// TwinCAT 3 PLC project SubSysPLC
// ProgramVersion: 3.1.4022.7
// libraries:
//   Tc2_MC2, * (Beckhoff Automation GmbH)
//   Tc2_Standard, * (Beckhoff Automation GmbH)
//   Tc2_System, * (Beckhoff Automation GmbH)
//   Tc2_Utilities, * (Beckhoff Automation GmbH)
//   Tc3_Module, * (Beckhoff Automation GmbH)
//   PMPS,0.0.0,SLAC - LCLS
// project tree:
//   DUTs/ ST_BinarySolidAttenuator.TcDUT, ST_SolidAttenuatorBlade.TcDUT
//   GVLs/ GVL.TcGVL
//   / PlcTask.TcTTO
//   POUs/DatabaseComponents/ FB_ExampleDeviceSM_DB.TcPOU, FB_MySQL_Client.TcPOU, F_DB_To_hTable.TcPOU
//   POUs/DeviceImplementationEx1/ FB_ExampleDevice.TcPOU, FB_ExampleDeviceSM.TcPOU
//   POUs/DeviceImplementationEx2/ FB_DevMover.TcPOU, FB_ExampleDeviceSM_All.TcPOU
//   POUs/ Fast_Faults_Evaluate.TcPOU, MAIN.TcPOU, PMPS.TcPOU
// real-time tasks:
//   TASK PlcTask: cycle T#10ms, priority 20, ADS port 350
// motion (NC):
//   TASK NC-Task 1 SAF: cycle T#2ms, priority 4, ADS port 501
//   TASK NC-Task 1 SVB: cycle T#10ms, priority 8, ADS port 511
//   AXIS DevRunner_1 (id 3)
//     OtherSettings: AllowMotionCmdToSlave=true
//     encoder EncType=1
//     drive DrvType=5
//       Analog: ScaleFactorActTorque=0.1
//     controller CtrType=1
//       CtrPara: PriorControlFactor=1
//         Observer: BandWidth=20
//   AXIS DevRunner_2 (id 4)
//     OtherSettings: AllowMotionCmdToSlave=true
//     encoder EncType=1
//     drive DrvType=5
//       Analog: ScaleFactorActTorque=0.1
//     controller CtrType=1
//       CtrPara: PriorControlFactor=1
//         Observer: BandWidth=20
//   AXIS DevRunner_3 (id 5)
//     OtherSettings: AllowMotionCmdToSlave=true
//     encoder EncType=1
//     drive DrvType=5
//       Analog: ScaleFactorActTorque=0.1
//     controller CtrType=1
//       CtrPara: PriorControlFactor=1
//         Observer: BandWidth=20
//   AXIS DevRunner_4 (id 6)
//     OtherSettings: AllowMotionCmdToSlave=true
//     encoder EncType=1
//     drive DrvType=5
//       Analog: ScaleFactorActTorque=0.1
//     controller CtrType=1
//       CtrPara: PriorControlFactor=1
//         Observer: BandWidth=20
//   AXIS DevRunner_5 (id 7)
//     OtherSettings: AllowMotionCmdToSlave=true
//     encoder EncType=1
//     drive DrvType=5
//       Analog: ScaleFactorActTorque=0.1
//     controller CtrType=1
//       CtrPara: PriorControlFactor=1
//         Observer: BandWidth=20
//   AXIS DevRunner_6 (id 8)
//     OtherSettings: AllowMotionCmdToSlave=true
//     encoder EncType=1
//     drive DrvType=5
//       Analog: ScaleFactorActTorque=0.1
//     controller CtrType=1
//       CtrPara: PriorControlFactor=1
//         Observer: BandWidth=20
//   AXIS DevRunner_7 (id 9)
//     OtherSettings: AllowMotionCmdToSlave=true
//     encoder EncType=1
//     drive DrvType=5
//       Analog: ScaleFactorActTorque=0.1
//     controller CtrType=1
//       CtrPara: PriorControlFactor=1
//         Observer: BandWidth=20
//   AXIS DevRunner_8 (id 10)
//     OtherSettings: AllowMotionCmdToSlave=true
//     encoder EncType=1
//     drive DrvType=5
//       Analog: ScaleFactorActTorque=0.1
//     controller CtrType=1
//       CtrPara: PriorControlFactor=1
//         Observer: BandWidth=20
//   AXIS Dev1 (id 1)
//     OtherSettings: AllowMotionCmdToSlave=true
//     encoder EncType=1
//     drive DrvType=5
//       Analog: ScaleFactorActTorque=0.1
//     controller CtrType=1
//       CtrPara: PriorControlFactor=1
//         Observer: BandWidth=20
//   AXIS Dev2 (id 2)
//     OtherSettings: AllowMotionCmdToSlave=true
//     encoder EncType=1
//     drive DrvType=5
//       Analog: ScaleFactorActTorque=0.1
//     controller CtrType=1
//       CtrPara: PriorControlFactor=1
//         Observer: BandWidth=20
// I/O:
//   DEVICE Device 1 (EtherCAT), AmsNetId 0.0.0.0.2.1
//     Term 3 (EK1200) [EK1200-5000 EtherCAT Power supply (2A E-Bus)]
//       PMPS_FFO [EL2202 2Ch. Dig. Output 24V, 0.5A]
//       PMPS_PRE [EL6692 EtherCAT Bridge terminal (Primary)]
// variable links:
//   SubSysPLC Instance <-> Device 1 (EtherCAT)/Term 3 (EK1200)/PMPS_FFO
//     PlcTask Outputs/GVL.g_FastFaultOutput1.q_xFastFaultOut <-> Channel 1/Output
//   SubSysPLC Instance <-> Device 1 (EtherCAT)/Term 3 (EK1200)/PMPS_PRE
//     PlcTask Inputs/PMPS.fbArbiterIO.i_stCurrentBP <-> IO Inputs/CurrentBP
//     PlcTask Inputs/PMPS.fbArbiterIO.xTxPDO_state <-> SYNC Inputs/TxPDO state
//     PlcTask Inputs/PMPS.fbArbiterIO.xTxPDO_toggle <-> SYNC Inputs/TxPDO toggle
//     PlcTask Outputs/PMPS.fbArbiterIO.q_stRequestedBP <-> IO Outputs/RequestedBP
//   SubSysPLC Instance <-> NC-Task 1 SAF/Axes/Dev1
//     PlcTask Inputs/MAIN.fbDev1.stDevice.stAxis.NcToPlc <-> Outputs/ToPlc
//     PlcTask Outputs/MAIN.fbDev1.stDevice.stAxis.PlcToNc <-> Inputs/FromPlc
//   SubSysPLC Instance <-> NC-Task 1 SAF/Axes/Dev2
//     PlcTask Inputs/MAIN.fbDev2.stDevice.stAxis.NcToPlc <-> Outputs/ToPlc
//     PlcTask Outputs/MAIN.fbDev2.stDevice.stAxis.PlcToNc <-> Inputs/FromPlc
//   SubSysPLC Instance <-> NC-Task 1 SAF/Axes/DevRunner_1
//     PlcTask Inputs/MAIN.DevArray[1].stDevice.stAxis.NcToPlc <-> Outputs/ToPlc
//     PlcTask Outputs/MAIN.DevArray[1].stDevice.stAxis.PlcToNc <-> Inputs/FromPlc
//   SubSysPLC Instance <-> NC-Task 1 SAF/Axes/DevRunner_2
//     PlcTask Inputs/MAIN.DevArray[2].stDevice.stAxis.NcToPlc <-> Outputs/ToPlc
//     PlcTask Outputs/MAIN.DevArray[2].stDevice.stAxis.PlcToNc <-> Inputs/FromPlc
//   SubSysPLC Instance <-> NC-Task 1 SAF/Axes/DevRunner_3
//     PlcTask Inputs/MAIN.DevArray[3].stDevice.stAxis.NcToPlc <-> Outputs/ToPlc
//     PlcTask Outputs/MAIN.DevArray[3].stDevice.stAxis.PlcToNc <-> Inputs/FromPlc
//   SubSysPLC Instance <-> NC-Task 1 SAF/Axes/DevRunner_4
//     PlcTask Inputs/MAIN.DevArray[4].stDevice.stAxis.NcToPlc <-> Outputs/ToPlc
//     PlcTask Outputs/MAIN.DevArray[4].stDevice.stAxis.PlcToNc <-> Inputs/FromPlc
//   SubSysPLC Instance <-> NC-Task 1 SAF/Axes/DevRunner_5
//     PlcTask Inputs/MAIN.DevArray[5].stDevice.stAxis.NcToPlc <-> Outputs/ToPlc
//     PlcTask Outputs/MAIN.DevArray[5].stDevice.stAxis.PlcToNc <-> Inputs/FromPlc
//   SubSysPLC Instance <-> NC-Task 1 SAF/Axes/DevRunner_6
//     PlcTask Inputs/MAIN.DevArray[6].stDevice.stAxis.NcToPlc <-> Outputs/ToPlc
//     PlcTask Outputs/MAIN.DevArray[6].stDevice.stAxis.PlcToNc <-> Inputs/FromPlc
//   SubSysPLC Instance <-> NC-Task 1 SAF/Axes/DevRunner_7
//     PlcTask Inputs/MAIN.DevArray[7].stDevice.stAxis.NcToPlc <-> Outputs/ToPlc
//     PlcTask Outputs/MAIN.DevArray[7].stDevice.stAxis.PlcToNc <-> Inputs/FromPlc
//   SubSysPLC Instance <-> NC-Task 1 SAF/Axes/DevRunner_8
//     PlcTask Inputs/MAIN.DevArray[8].stDevice.stAxis.NcToPlc <-> Outputs/ToPlc
//     PlcTask Outputs/MAIN.DevArray[8].stDevice.stAxis.PlcToNc <-> Inputs/FromPlc

CONFIGURATION SubSysPLC
    RESOURCE PLC ON TwinCAT3
        TASK PlcTask(INTERVAL := T#10ms, PRIORITY := 20);
        PROGRAM MAIN WITH PlcTask : MAIN;
    END_RESOURCE
END_CONFIGURATION

// ---- DUTs/ST_BinarySolidAttenuator.TcDUT
TYPE ST_BinarySolidAttenuator :
STRUCT
	axBlades	: ARRAY [0..9] OF ST_SolidAttenuatorBlade;
END_STRUCT
END_TYPE

// ---- DUTs/ST_SolidAttenuatorBlade.TcDUT
TYPE ST_SolidAttenuatorBlade :
STRUCT
	xRequestedIn	:	BOOL;
	xCurrentIn	:	BOOL;
	rThickness	:	REAL;
END_STRUCT
END_TYPE

// ---- GVLs/GVL.TcGVL

VAR_GLOBAL
	g_fbArbiter1	:	FB_Arbiter;
	g_fbArbiter2	:	FB_Arbiter;
	{attribute 'TcLinkTo' := '.q_xFastFaultOut:=TIIB[PMPS_FFO]^Channel 1^Output'}
	g_FastFaultOutput1	:	FB_HardwareFFOutput;
	g_rTestingVelocity	:	LREAL := PMPS_GVL.VISIBLE_TEST_VELOCITY;
END_VAR

// ---- POUs/MAIN.TcPOU
PROGRAM MAIN
VAR
	fbDev1	:	FB_ExampleDeviceSM_All;
	fbDev1Mover	:	FB_DevMover;
	fbDev2	:	FB_ExampleDeviceSM_All;
	fbDev2Mover	:	FB_DevMover;
	
	rtInit	:	R_TRIG;
	Initialize	:	BOOL := TRUE;
	
	DevArray : ARRAY[1..8] OF FB_ExampleDeviceSM_All;
	DevMoverArray : ARRAY [1..8] OF FB_DevMover;
	
	//fbDev3	:	FB_ExampleDeviceSM_DB;

	DevRunnerInt: INT;
	
	AttemptReset	:	TON;
    
    ffArray : ARRAY[1..FF_ARRAY] OF FB_FastFault;
    FFRunnerInt : INT := 1;
END_VAR
VAR CONSTANT
    FF_ARRAY : INT := 200;
END_VAR

//Sub-system Device PLC

IF Initialize THEN
	fbDev1(cBase := 10,
		fbFastFaultOutput := g_FastFaultOutput1,
		fbArbiter := g_fbArbiter1);
	fbDev2(cBase := 1000,
		fbFastFaultOutput := g_FastFaultOutput1,
		fbArbiter := g_fbArbiter1);
	g_fbArbiter1.A_Init();

//	fbDev3(cBase := 0,iDBID:=1,sDBNetId:='172.21.42.53.1.1',sDeviceID:='1',
//		fbArbiter := g_fbArbiter,
//		fbFastFaultOutput := g_FastFaultOutput1);

	FOR DevRunnerInt := 1 TO 8 DO
		DevArray[DevRunnerInt](cBase := DevRunnerInt*1000,
			fbFastFaultOutput := g_FastFaultOutput1,
			fbArbiter := g_fbArbiter1);
	END_FOR

	Initialize := FALSE;
END_IF

//Example devices
fbDev1(fbFastFaultOutput := g_FastFaultOutput1,
		fbArbiter := g_fbArbiter1);
fbDev2(fbFastFaultOutput := g_FastFaultOutput1,
		fbArbiter := g_fbArbiter1);
		
fbDev1Mover(Device:=fbDev1.stDevice);
fbDev2Mover(Device:=fbDev2.stDevice);

FOR DevRunnerInt := 1 TO 8 DO
	DevArray[DevRunnerInt](cBase := DevRunnerInt*1000,
		fbFastFaultOutput := g_FastFaultOutput1,
		fbArbiter := g_fbArbiter1);
		
	DevMoverArray[DevRunnerInt](Device := DevArray[DevRunnerInt].stDevice);	
END_FOR
(*
FOR FFRunnerInt := 1 to FF_ARRAY DO
    ffArray[FFRunnerInt](io_fbFFHWO := g_FastFaultOutput1);
END_FOR
*)		
PMPS();

Fast_Faults_Evaluate();

ACTION Initialize:

END_ACTION

END_PROGRAM

// ---- POUs/DeviceImplementationEx2/FB_ExampleDeviceSM_All.TcPOU
(* This version of the block is self contained. Minimizes wiring.*)
FUNCTION_BLOCK FB_ExampleDeviceSM_All
VAR_INPUT
	cBase: UDINT;
END_VAR
VAR_OUTPUT
END_VAR
VAR_IN_OUT
	fbFastFaultOutput	:	FB_HardwareFFOutput;
	fbArbiter	:	FB_Arbiter;
END_VAR
VAR
	stDevice	:	ST_Device;
	fbGovernor	:	FB_LinearGovernor;
	mcPower	:	MC_Power;
	mcStop: MC_Stop;
	mcAbsolute	:	MC_MoveAbsolute;
	fbBPTM	:	BeamParameterTransitionManager;
	xStartMove: BOOL;
	
	stCheckState: ST_DeviceState;
	stTargetState	:	ST_DeviceState; //Target device state

END_VAR
VAR PERSISTENT
	nLastActiveState	:	UDINT;
END_VAR

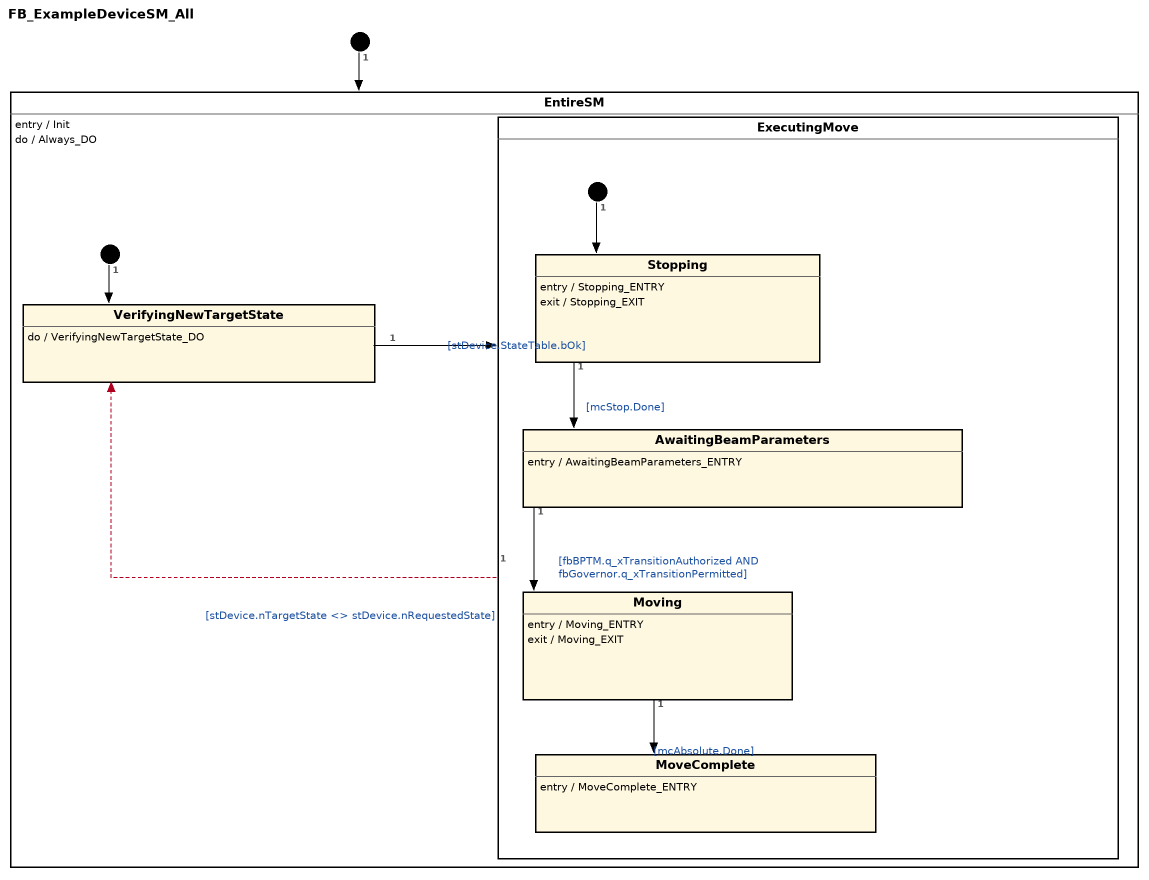
STATECHART FB_ExampleDeviceSM_All_1  // abortable
    START StartState3
    COMPOSITE STATE EntireSM
        entry / Init
        do / Always_DO
        START StartState1
        COMPOSITE STATE ExecutingMove
            START StartState2
            STATE Stopping
                entry / Stopping_ENTRY
                exit / Stopping_EXIT
            STATE AwaitingBeamParameters
                entry / AwaitingBeamParameters_ENTRY
            STATE Moving
                entry / Moving_ENTRY
                exit / Moving_EXIT
            STATE MoveComplete
                entry / MoveComplete_ENTRY
            StartState2 -> Stopping  // priority 1, on completion
            Stopping -> AwaitingBeamParameters [mcStop.Done] // priority 1, rising edge
            AwaitingBeamParameters -> Moving [fbBPTM.q_xTransitionAuthorized AND fbGovernor.q_xTransitionPermitted] // priority 1, rising edge
            Moving -> MoveComplete [mcAbsolute.Done] // priority 1, rising edge
        END_STATE
        STATE VerifyingNewTargetState
            do / VerifyingNewTargetState_DO
        StartState1 -> VerifyingNewTargetState  // priority 1, on completion
        ExecutingMove -> VerifyingNewTargetState [stDevice.nTargetState <> stDevice.nRequestedState] // priority 1, exception, rising edge
        VerifyingNewTargetState -> ExecutingMove [stDevice.StateTable.bOk] // priority 1
    END_STATE
    StartState3 -> EntireSM  // priority 1, on completion
END_STATECHART

ACTION Always_DO:
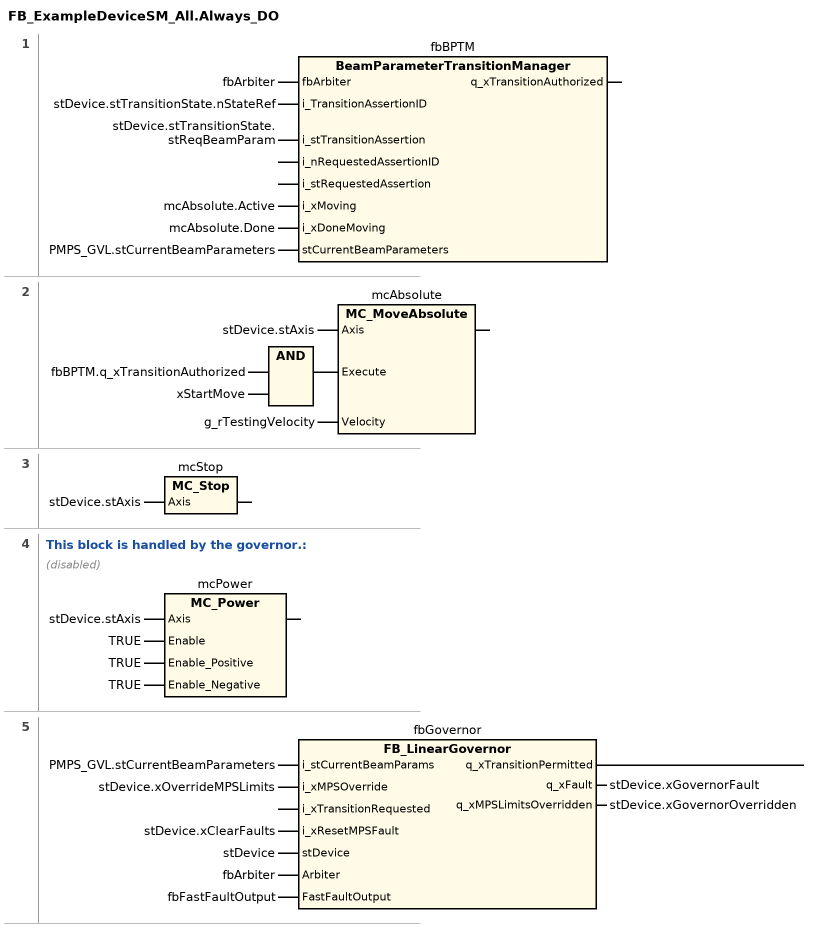
// NETWORK 1
fbBPTM(
    fbArbiter := fbArbiter,
    i_TransitionAssertionID := stDevice.stTransitionState.nStateRef,
    i_stTransitionAssertion := stDevice.stTransitionState.stReqBeamParam,
    i_xMoving := mcAbsolute.Active,
    i_xDoneMoving := mcAbsolute.Done,
    stCurrentBeamParameters := PMPS_GVL.stCurrentBeamParameters); // BeamParameterTransitionManager

// NETWORK 2
mcAbsolute(
    Axis := stDevice.stAxis,
    Execute := fbBPTM.q_xTransitionAuthorized AND xStartMove,
    Velocity := g_rTestingVelocity); // MC_MoveAbsolute

// NETWORK 3
mcStop(Axis := stDevice.stAxis); // MC_Stop

// NETWORK 4 (disabled)
// label: This block is handled by the governor.
// mcPower(Axis := stDevice.stAxis, Enable := TRUE, Enable_Positive := TRUE, Enable_Negative := TRUE); // MC_Power

// NETWORK 5
fbGovernor(
    i_stCurrentBeamParams := PMPS_GVL.stCurrentBeamParameters,
    i_xMPSOverride := stDevice.xOverrideMPSLimits,
    i_xResetMPSFault := stDevice.xClearFaults,
    stDevice := stDevice,
    Arbiter := fbArbiter,
    FastFaultOutput := fbFastFaultOutput,
    q_xFault => stDevice.xGovernorFault,
    q_xMPSLimitsOverridden => stDevice.xGovernorOverridden); // FB_LinearGovernor
END_ACTION

ACTION AwaitingBeamParameters_ENTRY:
fbBPTM.i_stRequestedAssertion := stTargetState.stReqBeamParam;
fbBPTM.i_nRequestedAssertionID := stTargetState.nStateRef;

//Tell the governor that we're trying to move.
fbGovernor.i_xTransitionRequested := TRUE;
END_ACTION

ACTION Init:

//Safe State
stDevice.nSafeState := cBase;
stDevice.nTransitionState := cBase+100;

//Initialize the State Table
stDevice.StateTable.A_Reset();

//Device State Table Instantiation
//To be done by the device state table database system
F_SetStateParams(
	nStateRef := stDevice.nSafeState,
	rPosition := 0,
	rTolerance := 10,
	stBeamParams := PMPS_GVL.cstFullBeam,
	Table := stDevice.StateTable
);
F_SetStateParams(
	nStateRef := cBase + 1,
	rPosition := 100,
	rTolerance := 10,
	stBeamParams := F_SetBeamParams(
		fAtt := 20,
		fPP_mJ := 1,
		neVRange	:= 2#1111_1011_1111_0000,
		nRate := 10
		),
	Table := stDevice.StateTable
);
F_SetStateParams(
	nStateRef := cBase + 2,
	rPosition := 200,
	rTolerance := 10,
	stBeamParams := F_SetBeamParams(
		fAtt := 30,
		fPP_mJ := 1,
		neVRange	:= 2#1111_1011_1111_0000,
		nRate := 10
		),
	Table := stDevice.StateTable
);
F_SetStateParams(
	nStateRef := cBase + 3,
	rPosition := 300,
	rTolerance := 10,
	stBeamParams := F_SetBeamParams(
		fAtt := 20,
		fPP_mJ := 1,
		neVRange	:= 2#1111_1011_1111_0000,
		nRate := 10
		),
	Table := stDevice.StateTable
);

F_SetStateParams(
	nStateRef := stDevice.nTransitionState,
	rPosition := 0,
	rTolerance := 0,
	stBeamParams := F_SetBeamParams(
		fAtt := 0,
		fPP_mJ := 0,
		neVRange	:= 2#1111_1011_1111_0000,
		nRate := 0
		),
	Table := stDevice.StateTable
);

//Set device transition state
stDevice.StateTable.A_Lookup(
	key := stDevice.nTransitionState,
	getValue => stDevice.stTransitionState
);

//Need an initialization routine for setting the active state
//Check if the device is at safe state
//If the device is within the state boundaries, it's considered to be in that state
stDevice.StateTable.A_Lookup(key:= stDevice.nSafeState);
IF stDevice.StateTable.bOk THEN
	stCheckState := stDevice.StateTable.getValue;
ELSE
	stCheckState := stDevice.stTransitionState; //This needs to be safer <TODO>
END_IF

IF stDevice.stAxis.NcToPlc.ActPos <= stCheckstate.rPosition + stCheckState.rTolerance AND
	stDevice.stAxis.NcToPlc.ActPos >= stCheckState.rPosition - stCheckState.rTolerance THEN
	stDevice.nActiveState := nLastActiveState;
ELSE
	stDevice.nActiveState := stDevice.nTransitionState;
END_IF

//Simulation Hardware Limit Switches
stDevice.i_xHiLim := TRUE;
stDevice.i_xLoLim := TRUE;
END_ACTION

ACTION MoveComplete_ENTRY:
//Clear transition request
fbGovernor.i_xTransitionRequested := FALSE;
//Latch active state
stDevice.nActiveState := stDevice.nTargetState;
nLastActiveState := stDevice.nActiveState;
END_ACTION

ACTION Moving_ENTRY:
xStartMove := TRUE;
mcAbsolute.Position := stTargetState.rPosition;
END_ACTION

ACTION Moving_EXIT:
xStartMove := FALSE;
END_ACTION

ACTION NewMove_ENTRY:

END_ACTION

ACTION Stopping_ENTRY:
mcStop.Execute := TRUE;
END_ACTION

ACTION Stopping_EXIT:
mcStop.Execute := FALSE;
END_ACTION

ACTION VerifyingNewTargetState_DO:
stDevice.StateTable.A_Lookup(
	key := stDevice.nRequestedState
);

IF stDevice.StateTable.bOk THEN
	stTargetState := stDevice.StateTable.getValue;
	stDevice.nTargetState := stDevice.nRequestedState;
ELSE
	; //log ignored state/ generate an error? <TODO>
END_IF
END_ACTION

END_FUNCTION_BLOCK

// ---- POUs/DeviceImplementationEx2/FB_DevMover.TcPOU
FUNCTION_BLOCK FB_DevMover
VAR_IN_OUT
	Device: ST_Device;
END_VAR

VAR
	DevMoverState: INT := 0;
	getPosPtr    : POINTER TO PMPS.T_HashTableEntry := 0;(* Returned hash table entry position pointer *)
	Pause : TON := (PT := T#5s);
	StartAgain: R_TRIG;
	Restart: BOOL;
END_VAR


StartAgain(CLK:=Restart);
Restart R= StartAgain.Q;
IF StartAgain.Q THEN
	DevMoverState := 0;
END_IF

CASE DevMoverState OF
	0:
		DevMoverState := 100;
	100: //Go to first entry in the state table
		Device.StateTable.A_GetFirst();
		//Device.nRequestedState := Device.StateTable.getValue.nStateRef;
		getPosPtr := Device.StateTable.getPosPtr;
		// Wait for move to complete
		DevMoverState := 300;
		
	200: // Wait for move
		
		// Once move is done, go to next entry in state table
		Pause(IN := Device.nActiveState = Device.nTargetState);
		IF Pause.Q THEN
			DevMoverState := 300;
		END_IF
(*		
	250: // Move to upper limit
	
	251: // Move to lower limit
*)	
	300: // Go to next entry
		Device.StateTable.A_GetNext(putPosPtr:=getPosPtr);
		
		// Go back to wait for move unless there are no more entries
		IF Device.StateTable.bOk AND (Device.StateTable.getValue.nStateRef <> Device.nRequestedState) THEN
			Device.nRequestedState := Device.StateTable.getValue.nStateRef;
			getPosPtr := Device.StateTable.getPosPtr;
			DevMoverState := 200;
		ELSE
			DevMoverState := 100;
		END_IF
		
	
END_CASE

END_FUNCTION_BLOCK

// ---- POUs/PMPS.TcPOU
PROGRAM PMPS
VAR
    
    fbArbiterIO : FB_SubSysToArbiter_IO;
END_VAR

fbArbiterIO(Arbiter := GVL.g_fbArbiter1, fbFFHWO := GVL.g_FastFaultOutput1);

END_PROGRAM

// ---- POUs/Fast_Faults_Evaluate.TcPOU
PROGRAM Fast_Faults_Evaluate
VAR
END_VAR

g_FastFaultOutput1.EvaluateOutput();

END_PROGRAM

// ---- POUs/DatabaseComponents/FB_ExampleDeviceSM_DB.TcPOU
(* This version of the block is self contained. Minimizes wiring.*)
FUNCTION_BLOCK FB_ExampleDeviceSM_DB
VAR_INPUT
	cBase: UDINT;
	iDBID:UDINT;
	sDBNetId: STRING;
	sDeviceID: STRING;
END_VAR
VAR_OUTPUT
END_VAR
VAR_IN_OUT
	fbArbiter : FB_Arbiter;
	fbFastFaultOutput	:	FB_HardwareFFOutput;
END_VAR
VAR
	stDevice	:	ST_Device;
	fbGovernor	:	FB_LinearGovernor;
	mcPower	:	MC_Power;
	mcStop: MC_Stop;
	mcAbsolute	:	MC_MoveAbsolute;
	fbBPTM	:	BeamParameterTransitionManager;
	xStartMove: BOOL;
	
	stCheckState: ST_DeviceState;
	stTargetState	:	ST_DeviceState; //Target device state
	fbDBClient:FB_MySQL_Client;
	bInitReady: BOOL :=FALSE;
	//aStateTable : ARRAY[1..PMPS_GVL.MAX_DEVICE_STATES] OF ST_DeviceStateTable;

END_VAR
VAR PERSISTENT
	nLastActiveState	:	UDINT;
END_VAR

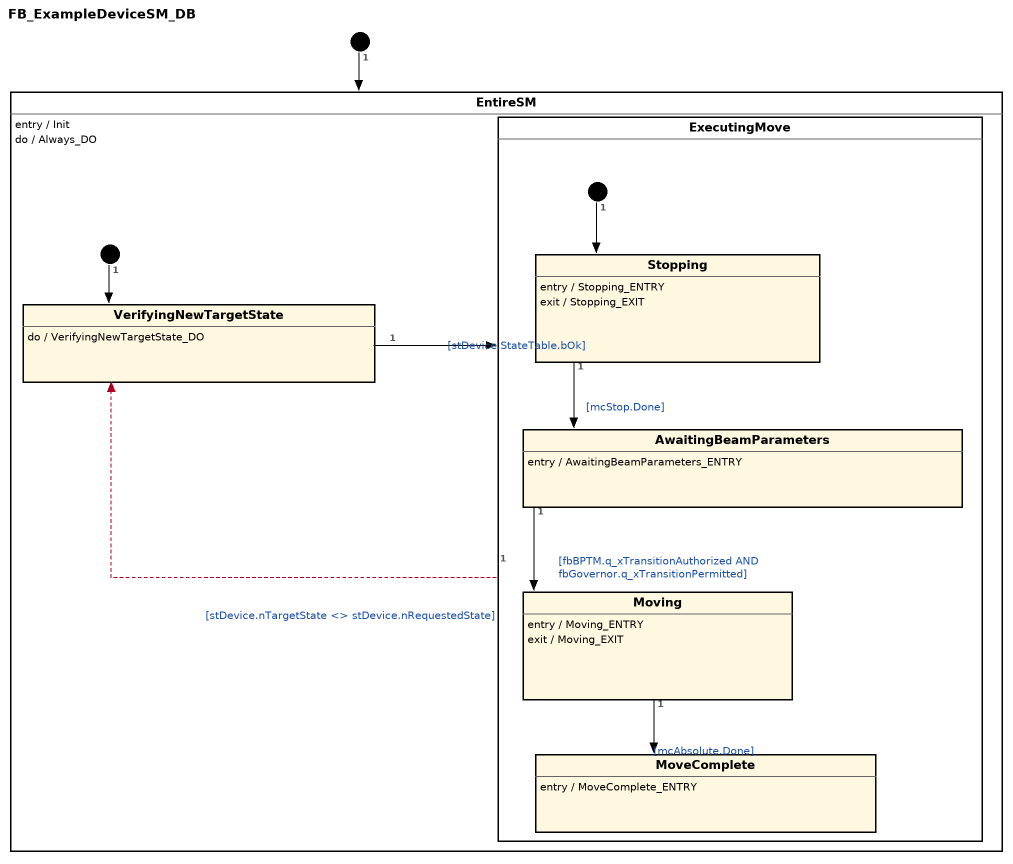
STATECHART FB_ExampleDeviceSM_DB  // abortable
    START StartState3
    COMPOSITE STATE EntireSM
        entry / Init
        do / Always_DO
        START StartState1
        COMPOSITE STATE ExecutingMove
            START StartState2
            STATE Stopping
                entry / Stopping_ENTRY
                exit / Stopping_EXIT
            STATE AwaitingBeamParameters
                entry / AwaitingBeamParameters_ENTRY
            STATE Moving
                entry / Moving_ENTRY
                exit / Moving_EXIT
            STATE MoveComplete
                entry / MoveComplete_ENTRY
            StartState2 -> Stopping  // priority 1, on completion
            Stopping -> AwaitingBeamParameters [mcStop.Done] // priority 1, rising edge
            AwaitingBeamParameters -> Moving [fbBPTM.q_xTransitionAuthorized AND fbGovernor.q_xTransitionPermitted] // priority 1, rising edge
            Moving -> MoveComplete [mcAbsolute.Done] // priority 1, rising edge
        END_STATE
        STATE VerifyingNewTargetState
            do / VerifyingNewTargetState_DO
        StartState1 -> VerifyingNewTargetState  // priority 1, on completion
        ExecutingMove -> VerifyingNewTargetState [stDevice.nTargetState <> stDevice.nRequestedState] // priority 1, exception, rising edge
        VerifyingNewTargetState -> ExecutingMove [stDevice.StateTable.bOk] // priority 1
    END_STATE
    StartState3 -> EntireSM  // priority 1, on completion
END_STATECHART

ACTION Always_DO:
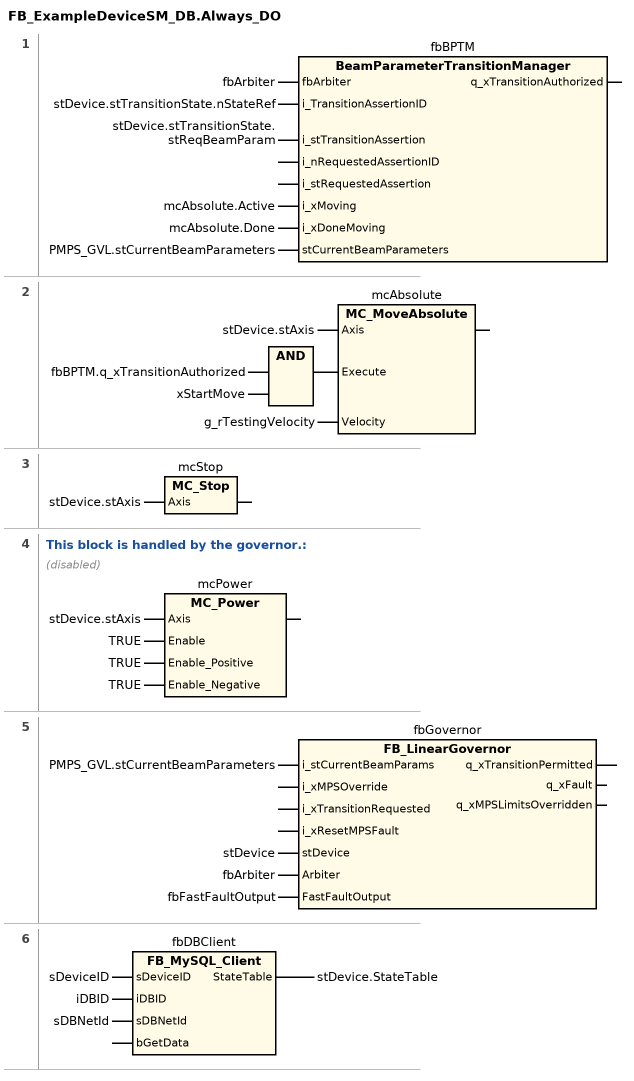
// NETWORK 1
fbBPTM(
    fbArbiter := fbArbiter,
    i_TransitionAssertionID := stDevice.stTransitionState.nStateRef,
    i_stTransitionAssertion := stDevice.stTransitionState.stReqBeamParam,
    i_xMoving := mcAbsolute.Active,
    i_xDoneMoving := mcAbsolute.Done,
    stCurrentBeamParameters := PMPS_GVL.stCurrentBeamParameters); // BeamParameterTransitionManager

// NETWORK 2
mcAbsolute(
    Axis := stDevice.stAxis,
    Execute := fbBPTM.q_xTransitionAuthorized AND xStartMove,
    Velocity := g_rTestingVelocity); // MC_MoveAbsolute

// NETWORK 3
mcStop(Axis := stDevice.stAxis); // MC_Stop

// NETWORK 4 (disabled)
// label: This block is handled by the governor.
// mcPower(Axis := stDevice.stAxis, Enable := TRUE, Enable_Positive := TRUE, Enable_Negative := TRUE); // MC_Power

// NETWORK 5
fbGovernor(
    i_stCurrentBeamParams := PMPS_GVL.stCurrentBeamParameters,
    stDevice := stDevice,
    Arbiter := fbArbiter,
    FastFaultOutput := fbFastFaultOutput); // FB_LinearGovernor

// NETWORK 6
fbDBClient(sDeviceID := sDeviceID, iDBID := iDBID, sDBNetId := sDBNetId); // FB_MySQL_Client
stDevice.StateTable := fbDBClient.StateTable;
END_ACTION

ACTION AwaitingBeamParameters_ENTRY:
fbBPTM.i_stRequestedAssertion := stTargetState.stReqBeamParam;
fbBPTM.i_nRequestedAssertionID := stTargetState.nStateRef;

//Tell the governor that we're trying to move.
fbGovernor.i_xTransitionRequested := TRUE;
END_ACTION

ACTION Init:
	
//Safe State
stDevice.nSafeState := cBase;
stDevice.nTransitionState := cBase+100;

//Initialize the State Table
stDevice.StateTable.A_Reset();
//Device State Table Instantiation
F_SetStateParams(
	nStateRef := stDevice.nSafeState,
	rPosition := 0,
	rTolerance := 10,
	stBeamParams := PMPS_GVL.cstFullBeam,
	Table := stDevice.StateTable
);
//Connect to DB and get state table data
fbDBClient.bGetData:= TRUE;//fbMySQL.nState:=400; 

stDevice.StateTable.A_Lookup(
		key := stDevice.nTransitionState,
		getValue => stDevice.stTransitionState
);
	
//Need an initialization routine for setting the active state
//Check if the device is at the last known state
//If the device is within the state boundaries, it's considered to be in that state
stDevice.StateTable.A_Lookup(key:= nLastActiveState);
IF stDevice.StateTable.bOk THEN
	stCheckState := stDevice.StateTable.getValue;
ELSE
	stCheckState := stDevice.stTransitionState; //This needs to be safer <TODO>
END_IF

IF stDevice.stAxis.NcToPlc.ActPos <= stCheckstate.rPosition + stCheckState.rTolerance AND
	stDevice.stAxis.NcToPlc.ActPos >= stCheckState.rPosition - stCheckState.rTolerance THEN
	stDevice.nActiveState := nLastActiveState;
ELSE
	stDevice.nActiveState := stDevice.nTransitionState;
END_IF

//Simulation Hardware Limit Switches
stDevice.i_xHiLim := TRUE;
stDevice.i_xLoLim := TRUE;
END_ACTION

ACTION Initialize:

END_ACTION

ACTION MoveComplete_ENTRY:
//Clear transition request
fbGovernor.i_xTransitionRequested := FALSE;
//Latch active state
stDevice.nActiveState := stDevice.nTargetState;
nLastActiveState := stDevice.nActiveState;
END_ACTION

ACTION Moving_ENTRY:
xStartMove := TRUE;
mcAbsolute.Position := stTargetState.rPosition;
END_ACTION

ACTION Moving_EXIT:
xStartMove := FALSE;
END_ACTION

ACTION NewMove_ENTRY:

END_ACTION

ACTION Stopping_ENTRY:
mcStop.Execute := TRUE;
END_ACTION

ACTION Stopping_EXIT:
mcStop.Execute := FALSE;
END_ACTION

ACTION VerifyingNewTargetState_DO:
stDevice.StateTable.A_Lookup(
	key := stDevice.nRequestedState
);

IF stDevice.StateTable.bOk THEN
	stTargetState := stDevice.StateTable.getValue;
	stDevice.nTargetState := stDevice.nRequestedState;
ELSE
	; //log ignored state/ generate an error? <TODO>
END_IF
END_ACTION

END_FUNCTION_BLOCK

// ---- POUs/DatabaseComponents/FB_MySQL_Client.TcPOU
FUNCTION_BLOCK FB_MySQL_Client
VAR_INPUT
	sDeviceID: STRING;
	iDBID:UDINT;
	sDBNetId: STRING ;
	bGetData:BOOL;
END_VAR
VAR_OUTPUT
	StateTable : FB_LinearDeviceStateTable;
END_VAR
VAR CONSTANT
	sSQLCommand :STRING:='SELECT * FROM device_states  WHERE device_id =';
END_VAR
VAR
	nState: INT:=0; // used as a start signal
	nRecordCount: UDINT:=PMPS_GVL.MAX_DEVICE_STATES;
	aDeviceStateTable : ARRAY[1..PMPS_GVL.MAX_DEVICE_STATES] OF ST_DeviceStateTable;
	fbMySQLDB:  FB_SQLDatabase(sNetId := '', tTimeout:=T#5S);
	fbSQLCmd:  FB_SQLCommand(sNetId := '', tTimeout:=T#5S);
	fbSQLResult: FB_SQLResult(sNetId := '', tTimeout:=T#5S);
	sSQLCmd :STRING;
	ipResultEvent : Tc3_Eventlogger.I_TcResultEvent;
	
	
END_VAR


IF (bGetData) THEN
	bGetData:= FALSE;
	nState := 100;
END_IF

CASE nState OF
	0:
100:// Initialize Database function blocks
	fbMySQLDB.sNetID := sDBNetId;
	fbSQLCmd.sNetID := sDBNetId;
	fbSQLResult.sNetID := sDBNetId; 
	IF fbMySQLDB.Connect(iDBID) THEN
		IF fbMySQLDB.bError THEN
			nState := 9000+nState; 
		ELSE
			nState := nState+1; 
		END_IF
	END_IF
 
101:	
	 IF(fbMySQLDB.bConnected ) THEN
		fbMySQLDB.CreateCmd(pSQLCommand := ADR(fbSQLCmd));
		IF fbMySQLDB.bError THEN
			nState := 9000+nState; 
		ELSE
			nState := 1+nState; 
		END_IF
	 END_IF
102:	 
  (*Execute SQL Comnmand*)
	//sSQLCmd :=sSQLCommand;
	sSQLCmd := CONCAT(sSQLCommand, sDeviceID) ;		
   IF fbSQLCmd.ExecuteDataReturn(pSQLCmd:=ADR(sSQLCmd),cbSQLCmd:=SIZEOF(sSQLCmd),pSQLDBResult:=ADR(fbSQLResult)) THEN
   	IF( fbSQLCmd.bError) THEN
	    nState := 9000+nState; 
    ELSE
        nState := 1+nState; 
		MEMSET(ADR(aDeviceStateTable),0,SIZEOF(aDeviceStateTable));

    END_IF
  END_IF
 
103: 
	(*Read data FROM the database*)
  IF (fbSQLResult.Read(nStartIndex:=0, nRecordCount:=nRecordCount,pData:=ADR(aDeviceStateTable),cbData:=SIZEOF(aDeviceStateTable),bWithVerifying:=TRUE,bDataRelease:=TRUE) )THEN
	 ipResultEvent := fbSQLResult.ipTcResultEvent;
	IF fbSQLResult.bError THEN
         nState := 9000+nState; 
    ELSE
        nState := 500;// 1+nState; 
    END_IF
END_IF	

500:
	//Device State Table Instantiation
	IF F_DB_To_hTable( aStatesParamsTable:= aDeviceStateTable, nRecordCount:=nRecordCount, Table := StateTable)THEN
         nState := 9000+nState; 
    ELSE
        nState :=800;// 1+nState; 
    END_IF



600: //Reload DATA
//Reset all hash table entries
// re instantiate device state table	
	;
9500:
800: //Release and Disconnect
	
	IF (fbSQLResult.Release() AND fbMySQLDB.Disconnect()) THEN
		nState:=-1;
		ELSE
			 nState := 9000+nState; 
	END_IF


		;
END_CASE

END_FUNCTION_BLOCK

// ---- POUs/DatabaseComponents/F_DB_To_hTable.TcPOU
FUNCTION F_DB_To_hTable : BOOL
VAR_INPUT
	aStatesParamsTable : ARRAY[1..PMPS_GVL.MAX_DEVICE_STATES] OF ST_DeviceStateTable;
	nRecordCount: UDINT;
END_VAR
VAR_IN_OUT
	Table	:	FB_LinearDeviceStateTable;
END_VAR
VAR
	stDeviceState	:	ST_DeviceState;
	iRow : UDINT:=1;
END_VAR

Table.A_Reset();
//Device State Table Instantiation
(*F_SetStateParams(
	nStateRef := 0,
	rPosition := 0,
	rTolerance := 0,
	stBeamParams := PMPS_GVL.cstFullBeam,
	Table := Table
);
*)
IF (nRecordCount>0) THEN
	FOR iRow:=1 TO nRecordCount BY 1 DO
	stDeviceState.nStateRef := DINT_TO_UDINT(aStatesParamsTable[iRow].iStateID);
	stDeviceState.rPosition := aStatesParamsTable[iRow].rTargetPosition;
	stDeviceState.rTolerance := aStatesParamsTable[iRow].rTolerance;  
	stDeviceState.stReqBeamParam.fAtt := aStatesParamsTable[iRow].rTransmission;
	stDeviceState.stReqBeamParam.fPP_mJ := (aStatesParamsTable[iRow].rPerPulseEnergy);
	stDeviceState.stReqBeamParam.nRate := DINT_TO_UDINT(aStatesParamsTable[iRow].iPulseRate);
	stDeviceState.stReqBeamParam.nBeamClass := DINT_TO_BYTE(aStatesParamsTable[iRow].iBeamClass);
//	stDeviceState.stReqBeamParam.fUpper_eV := (aStatesParamsTable[iRow].rUpper_eV);
//	stDeviceState.stReqBeamParam.fLower_eV := (aStatesParamsTable[iRow].rLower_eV);
	stDeviceState.stReqBeamParam.reV := aStatesParamsTable[iRow].rPhotonEnergy;
	//stDeviceState.stReqBeamParam.neVRange := (aStatesParamsTable[iRow].rLower_eV);
	Table.A_Add(
		key := stDeviceState.nStateRef,
		putValue := stDeviceState
	);
END_FOR;
END_IF

Table.A_Count();
F_DB_To_hTable := Table.bOk;

END_FUNCTION

// ---- POUs/DeviceImplementationEx1/FB_ExampleDevice.TcPOU
FUNCTION_BLOCK FB_ExampleDevice
VAR_INPUT
END_VAR
VAR_OUTPUT
END_VAR
VAR
	MC_MoveAbsolute_0: MC_MoveAbsolute;
	fbBCTM: BeamParameterTransitionManager;
	FB_ExampleDeviceSM_0: FB_ExampleDeviceSM;
	stDevice	:	ST_Device;
	MC_Power_0: MC_Power;
	MC_Stop_0	:	MC_Stop;
END_VAR

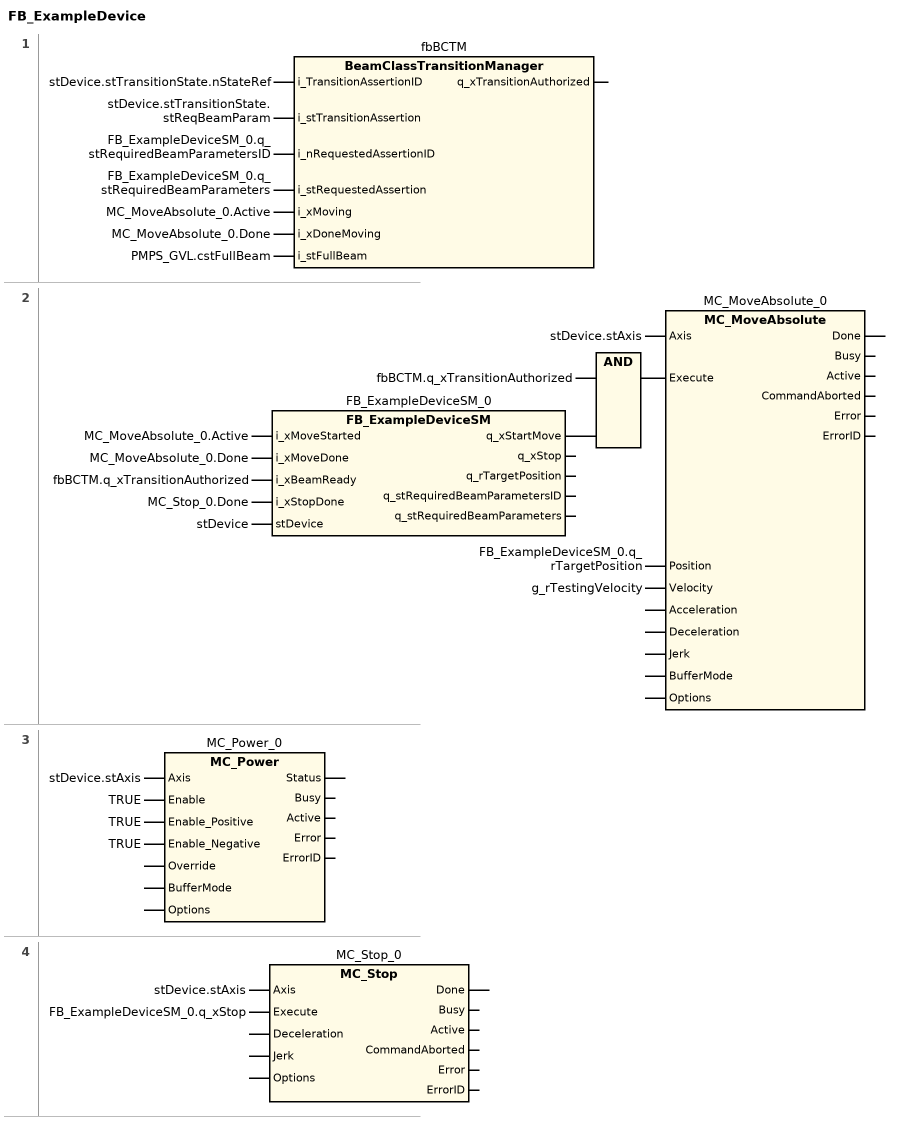
// NETWORK 1
fbBCTM(
    i_TransitionAssertionID := stDevice.stTransitionState.nStateRef,
    i_stTransitionAssertion := stDevice.stTransitionState.stReqBeamParam,
    i_nRequestedAssertionID := FB_ExampleDeviceSM_0.q_stRequiredBeamParametersID,
    i_stRequestedAssertion := FB_ExampleDeviceSM_0.q_stRequiredBeamParameters,
    i_xMoving := MC_MoveAbsolute_0.Active,
    i_xDoneMoving := MC_MoveAbsolute_0.Done,
    i_stFullBeam := PMPS_GVL.cstFullBeam); // BeamClassTransitionManager

// NETWORK 2
FB_ExampleDeviceSM_0(
    i_xMoveStarted := MC_MoveAbsolute_0.Active,
    i_xMoveDone := MC_MoveAbsolute_0.Done,
    i_xBeamReady := fbBCTM.q_xTransitionAuthorized,
    i_xStopDone := MC_Stop_0.Done,
    stDevice := stDevice); // FB_ExampleDeviceSM
MC_MoveAbsolute_0(
    Axis := stDevice.stAxis,
    Execute := fbBCTM.q_xTransitionAuthorized AND FB_ExampleDeviceSM_0.q_xStartMove,
    Position := FB_ExampleDeviceSM_0.q_rTargetPosition,
    Velocity := g_rTestingVelocity); // MC_MoveAbsolute

// NETWORK 3
MC_Power_0(Axis := stDevice.stAxis, Enable := TRUE, Enable_Positive := TRUE, Enable_Negative := TRUE); // MC_Power

// NETWORK 4
MC_Stop_0(Axis := stDevice.stAxis, Execute := FB_ExampleDeviceSM_0.q_xStop); // MC_Stop

ACTION Initialize:

stDevice.astStates[1].rPosition := 100;
stDevice.astStates[1].nStateRef := 16#1;
stDevice.astStates[1].stReqBeamParam := F_SetBeamParams(
	fAtt := 20,
	fPP_mJ := 1,
	fLower_eV := 0,
	fUpper_eV := 1500
);

stDevice.astStates[2].rPosition := 200;
stDevice.astStates[2].nStateRef := 16#2;
stDevice.astStates[2].stReqBeamParam := F_SetBeamParams(
	fAtt := 50,
	fPP_mJ := 1,
	fLower_eV := 0,
	fUpper_eV := 1500
);

stDevice.astStates[3].rPosition := 300;
stDevice.astStates[3].nStateRef := 16#3;
stDevice.astStates[3].stReqBeamParam := F_SetBeamParams(
	fAtt := 50,
	fPP_mJ := 0.5,
	fLower_eV := 0,
	fUpper_eV := 1500
);

stDevice.stTransitionState.nStateRef := 16#10;
stDevice.stTransitionState.stReqBeamParam := F_SetBeamParams(
	fAtt := 100,
	fPP_mJ := 1,
	fLower_eV := 0,
	fUpper_eV := 1500
);
END_ACTION

END_FUNCTION_BLOCK

// ---- POUs/DeviceImplementationEx1/FB_ExampleDeviceSM.TcPOU

FUNCTION_BLOCK FB_ExampleDeviceSM
VAR_INPUT
	i_xMoveStarted	:	BOOL; //Connect to moving flag
	i_xMoveDone	:	BOOL; //Connect to move done flag
	i_xBeamReady	:	BOOL; //Connect to transitioneer
	i_xStopDone	:	BOOL; //Connect to MC_Stop.Done
END_VAR
VAR_OUTPUT
	q_xStartMove	:	BOOL; //Connect to MC_Absolute.Execute
	q_xStop			:	BOOL; //Connect to MC_Stop.Execute
	q_rTargetPosition	:	REAL; //Connect to MC_Absolute.Position
	q_stRequiredBeamParametersID	:	UDINT;
	q_stRequiredBeamParameters	:	ST_BeamParams; //Connect to BeamParameterTransitionManager
END_VAR
VAR_IN_OUT
	stDevice	:	ST_Device;
END_VAR
VAR
	nTargetState	:	INT;
	
	xNewReq	:	BOOL; //Set true when new target request present
	
END_VAR

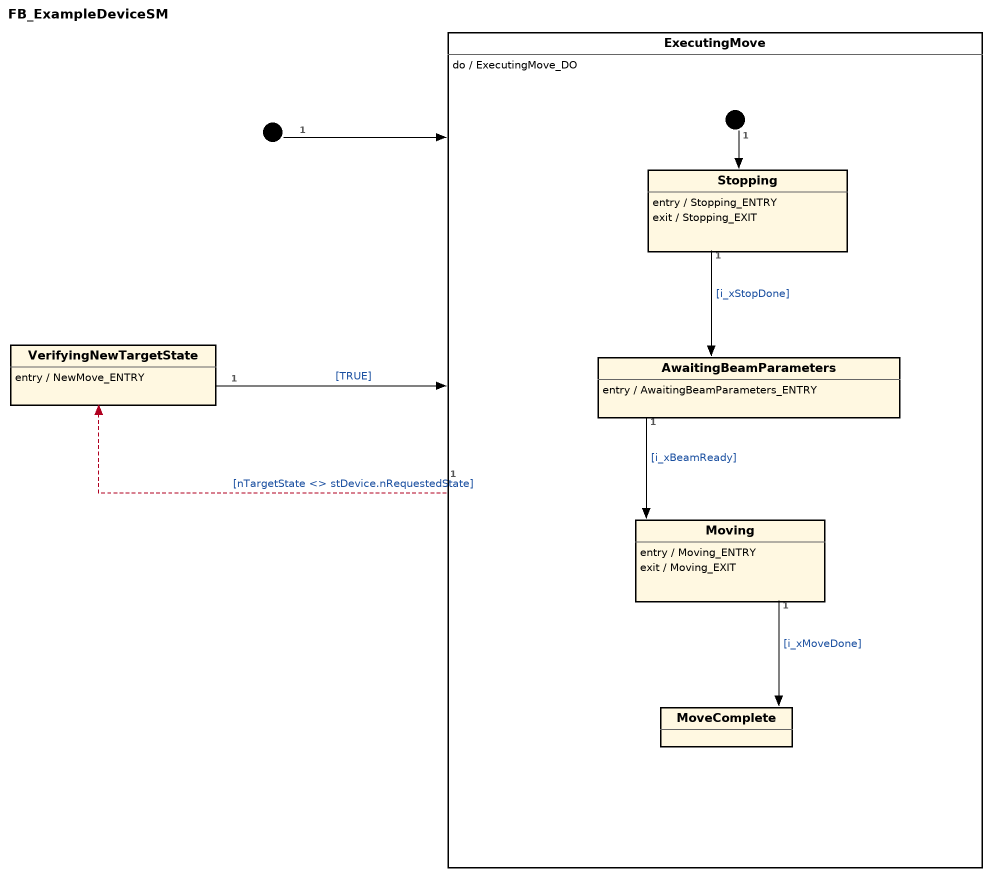
STATECHART FB_ExampleDeviceSM  // abortable
    START StartState1
    COMPOSITE STATE ExecutingMove
        do / ExecutingMove_DO
        START StartState2
        STATE Stopping
            entry / Stopping_ENTRY
            exit / Stopping_EXIT
        STATE AwaitingBeamParameters
            entry / AwaitingBeamParameters_ENTRY
        STATE Moving
            entry / Moving_ENTRY
            exit / Moving_EXIT
        STATE MoveComplete
        StartState2 -> Stopping  // priority 1, on completion
        Stopping -> AwaitingBeamParameters [i_xStopDone] // priority 1, rising edge
        AwaitingBeamParameters -> Moving [i_xBeamReady] // priority 1, rising edge
        Moving -> MoveComplete [i_xMoveDone] // priority 1, rising edge
    END_STATE
    STATE VerifyingNewTargetState
        entry / NewMove_ENTRY
    StartState1 -> ExecutingMove  // priority 1, on completion
    ExecutingMove -> VerifyingNewTargetState [nTargetState <> stDevice.nRequestedState] // priority 1, exception, rising edge
    VerifyingNewTargetState -> ExecutingMove [TRUE] // priority 1
END_STATECHART

ACTION AwaitingBeamParameters_ENTRY:
q_stRequiredBeamParameters := stDevice.astStates[nTargetState].stReqBeamParam;
q_stRequiredBeamParametersID := stDevice.astStates[nTargetState].nStateRef;
END_ACTION

ACTION ExecutingMove_DO:

END_ACTION

ACTION Moving_ENTRY:
q_xStartMove := TRUE;
q_rTargetPosition := stDevice.astStates[nTargetState].rPosition;
END_ACTION

ACTION Moving_EXIT:
q_xStartMove := FALSE;
END_ACTION

ACTION NewMove_ENTRY:

IF stDevice.nRequestedState <= PMPS_GVL.cnMaxStateArrayLen AND
	stDevice.nRequestedState >= 1 THEN
	nTargetState := stDevice.nRequestedState;
END_IF
END_ACTION

ACTION Stopping_ENTRY:
q_xStop	:= TRUE;
END_ACTION

ACTION Stopping_EXIT:
q_xStop := FALSE;
END_ACTION

END_FUNCTION_BLOCK
